PROGRAM Circuito_L4
VAR_INPUT
	Modo_Calibrar_L4: BOOL;
END_VAR
	
VAR
		fbBomba_L4 :Equipo_Motor_ATV320;
		ControlValv_ioLink_V1:ControlValv_ioLink;
		ControlValv_ioLink_V2: ControlValv_ioLink;
		ControlValv_ioLink_V3: ControlValv_ioLink;
		ControlValv_ioLink_V4: ControlValv_ioLink;
		Falla_L4_V1:BOOL;
		Falla_L4_V2:BOOL;
		Falla_L4_V3:BOOL;
		Falla_L4_V4:BOOL;
	Balanza_PU1_WT4: Balanza;
		dHS:DINT;
		TOF_calibradoIBC: TOF;
		TDemoraInyectar: TON;
		SetDemoraInyeccion: REAL;
	

	Volumen_L4: REAL;
	AuxVol: REAL;
	Total: REAL;
	auxIniCal: BOOL;
	Calculo_caudal_L4: Calculo_caudal;
	PID_L4_SP: REAL;
	PID_L4_PV: REAL;
	CorrecionCaudalxOffset_L4: CorrecionCaudalxOffset;
	tInyeccion: TON;
	PID_L4_manual: REAL;
	PID_L4: FB_PID;
	PID_L4_Kp: REAL := 0.1;
	PID_L4_Ti: REAL := 100;
	PID_L4_auto: BOOL;
	PID_L4_reset: BOOL;
	PID_L4_bMuerta: REAL := 5;
	Tiempo_seg_to_TIME_DemoraInyec: Tiempo_seg_to_TIME;
	AuxTDemoraInyec: TIME;
	Tiempo_TIME_to_seg_InyCal: Tiempo_TIME_to_seg;
	AuxInyCal:TIME;
	IniTotalFT2:REAL;
	Auxconsumo:REAL;
	ProductoAsociado: STRING;
	Lavagem_Circuito04: Lavagem;
	
END_VAR
VAR PERSISTENT
	UltimaCalibracao	:UDINT;	//Data e hora da ultima calibração
END_VAR
VAR // added by the converter: edge detectors and wires of the graphical bodies
    _w1, _w2, _w3, _w4, _w5, _w6, _w7, _w8, _w9, _w10, _w11, _w12, _w13 : BOOL;
    _ft1 : F_TRIG;
    _rt1, _rt2 : R_TRIG;
END_VAR

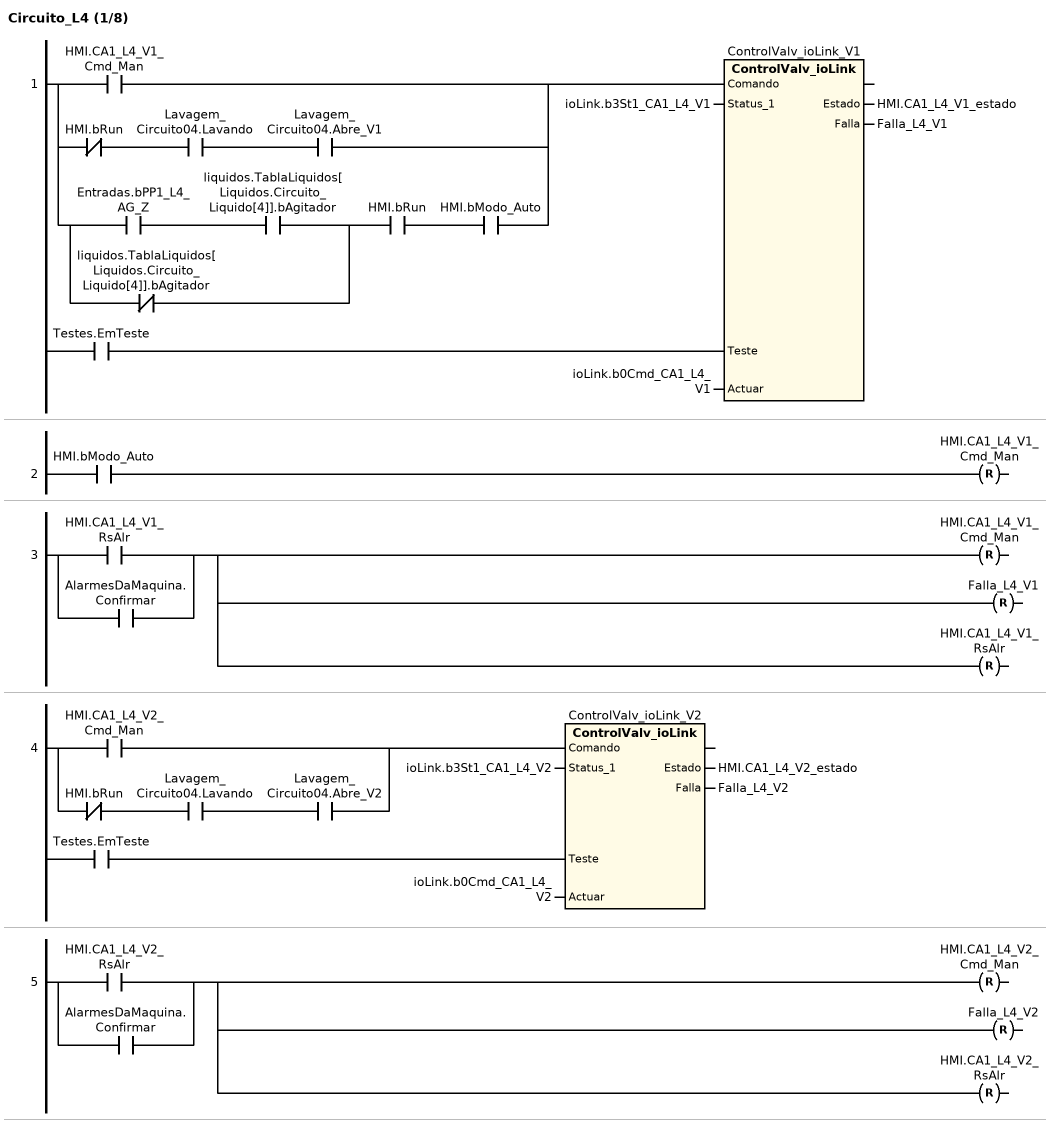
// NETWORK 1
ControlValv_ioLink_V1(
    Comando := HMI.CA1_L4_V1_Cmd_Man OR NOT HMI.bRun AND Lavagem_Circuito04.Lavando AND Lavagem_Circuito04.Abre_V1 OR (Entradas.bPP1_L4_AG_Z AND (liquidos.TablaLiquidos[Liquidos.Circuito_Liquido[4]].bAgitador) OR NOT (liquidos.TablaLiquidos[Liquidos.Circuito_Liquido[4]].bAgitador)) AND HMI.bRun AND HMI.bModo_Auto,
    Status_1 := ioLink.b3St1_CA1_L4_V1,
    Teste := Testes.EmTeste,
    Actuar := ioLink.b0Cmd_CA1_L4_V1,
    Estado => HMI.CA1_L4_V1_estado,
    Falla => Falla_L4_V1); // ControlValv_ioLink

// NETWORK 2
HMI.CA1_L4_V1_Cmd_Man R= HMI.bModo_Auto;

// NETWORK 3
_w1 := HMI.CA1_L4_V1_RsAlr OR AlarmesDaMaquina.Confirmar;
HMI.CA1_L4_V1_Cmd_Man R= _w1;
Falla_L4_V1 R= _w1;
HMI.CA1_L4_V1_RsAlr R= _w1;

// NETWORK 4
ControlValv_ioLink_V2(
    Comando := HMI.CA1_L4_V2_Cmd_Man OR NOT HMI.bRun AND Lavagem_Circuito04.Lavando AND Lavagem_Circuito04.Abre_V2,
    Status_1 := ioLink.b3St1_CA1_L4_V2,
    Teste := Testes.EmTeste,
    Actuar := ioLink.b0Cmd_CA1_L4_V2,
    Estado => HMI.CA1_L4_V2_estado,
    Falla => Falla_L4_V2); // ControlValv_ioLink

// NETWORK 5
_w2 := HMI.CA1_L4_V2_RsAlr OR AlarmesDaMaquina.Confirmar;
HMI.CA1_L4_V2_Cmd_Man R= _w2;
Falla_L4_V2 R= _w2;
HMI.CA1_L4_V2_RsAlr R= _w2;

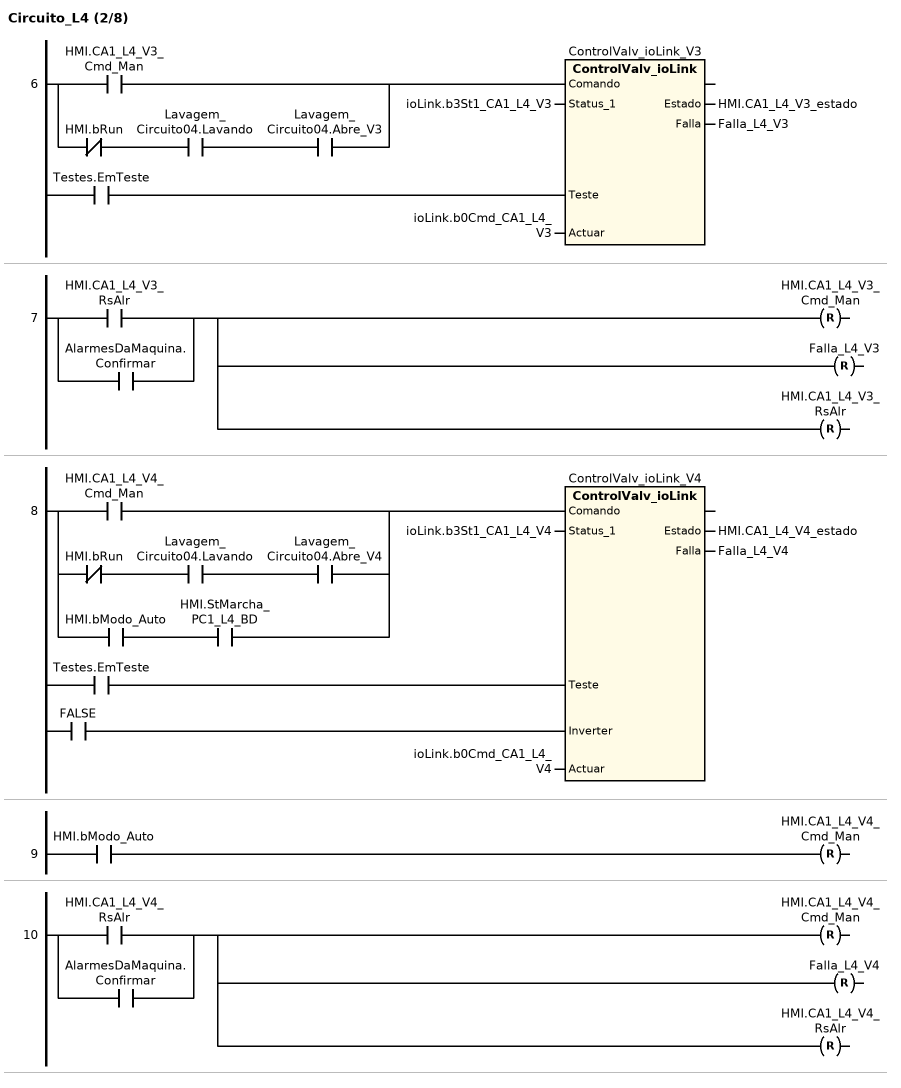
// NETWORK 6
ControlValv_ioLink_V3(
    Comando := HMI.CA1_L4_V3_Cmd_Man OR NOT HMI.bRun AND Lavagem_Circuito04.Lavando AND Lavagem_Circuito04.Abre_V3,
    Status_1 := ioLink.b3St1_CA1_L4_V3,
    Teste := Testes.EmTeste,
    Actuar := ioLink.b0Cmd_CA1_L4_V3,
    Estado => HMI.CA1_L4_V3_estado,
    Falla => Falla_L4_V3); // ControlValv_ioLink

// NETWORK 7
_w3 := HMI.CA1_L4_V3_RsAlr OR AlarmesDaMaquina.Confirmar;
HMI.CA1_L4_V3_Cmd_Man R= _w3;
Falla_L4_V3 R= _w3;
HMI.CA1_L4_V3_RsAlr R= _w3;

// NETWORK 8
ControlValv_ioLink_V4(
    Comando := HMI.CA1_L4_V4_Cmd_Man OR NOT HMI.bRun AND Lavagem_Circuito04.Lavando AND Lavagem_Circuito04.Abre_V4 OR HMI.bModo_Auto AND HMI.StMarcha_PC1_L4_BD,
    Status_1 := ioLink.b3St1_CA1_L4_V4,
    Teste := Testes.EmTeste,
    Inverter := FALSE,
    Actuar := ioLink.b0Cmd_CA1_L4_V4,
    Estado => HMI.CA1_L4_V4_estado,
    Falla => Falla_L4_V4); // ControlValv_ioLink

// NETWORK 9
HMI.CA1_L4_V4_Cmd_Man R= HMI.bModo_Auto;

// NETWORK 10
_w4 := HMI.CA1_L4_V4_RsAlr OR AlarmesDaMaquina.Confirmar;
HMI.CA1_L4_V4_Cmd_Man R= _w4;
Falla_L4_V4 R= _w4;
HMI.CA1_L4_V4_RsAlr R= _w4;

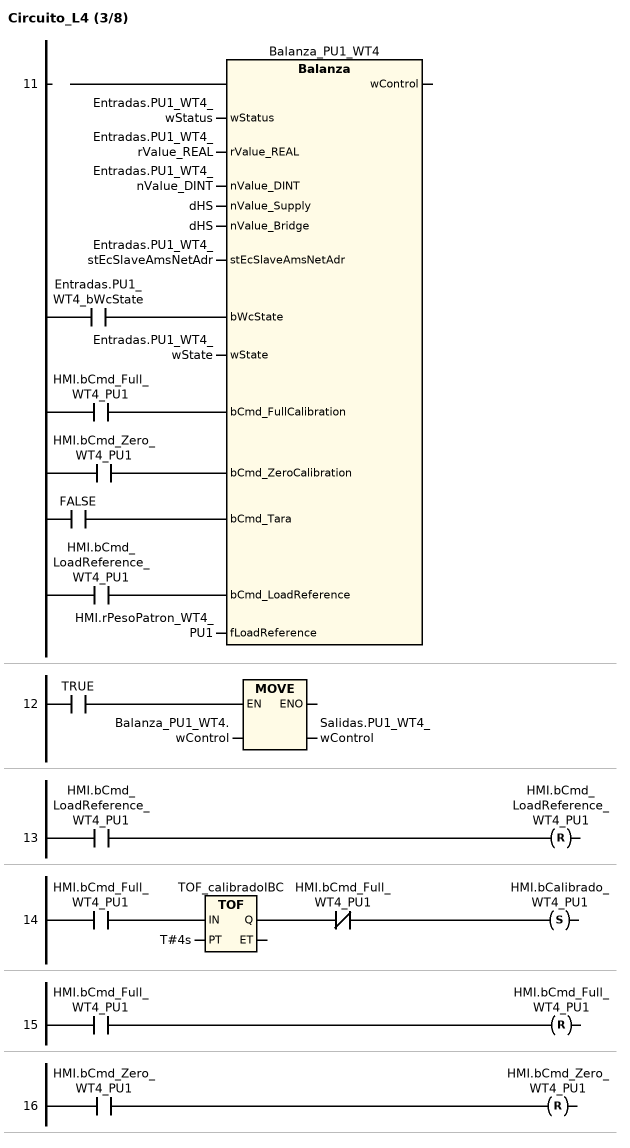
// NETWORK 11
Balanza_PU1_WT4(
    wStatus := Entradas.PU1_WT4_wStatus,
    rValue_REAL := Entradas.PU1_WT4_rValue_REAL,
    nValue_DINT := Entradas.PU1_WT4_nValue_DINT,
    nValue_Supply := dHS,
    nValue_Bridge := dHS,
    stEcSlaveAmsNetAdr := Entradas.PU1_WT4_stEcSlaveAmsNetAdr,
    bWcState := Entradas.PU1_WT4_bWcState,
    wState := Entradas.PU1_WT4_wState,
    bCmd_FullCalibration := HMI.bCmd_Full_WT4_PU1,
    bCmd_ZeroCalibration := HMI.bCmd_Zero_WT4_PU1,
    bCmd_Tara := FALSE,
    bCmd_LoadReference := HMI.bCmd_LoadReference_WT4_PU1,
    fLoadReference := HMI.rPesoPatron_WT4_PU1); // Balanza

// NETWORK 12
Salidas.PU1_WT4_wControl := Balanza_PU1_WT4.wControl;

// NETWORK 13
HMI.bCmd_LoadReference_WT4_PU1 R= HMI.bCmd_LoadReference_WT4_PU1;

// NETWORK 14
TOF_calibradoIBC(IN := HMI.bCmd_Full_WT4_PU1, PT := T#4s); // TOF
HMI.bCalibrado_WT4_PU1 S= TOF_calibradoIBC.Q AND NOT HMI.bCmd_Full_WT4_PU1;

// NETWORK 15
HMI.bCmd_Full_WT4_PU1 R= HMI.bCmd_Full_WT4_PU1;

// NETWORK 16
HMI.bCmd_Zero_WT4_PU1 R= HMI.bCmd_Zero_WT4_PU1;

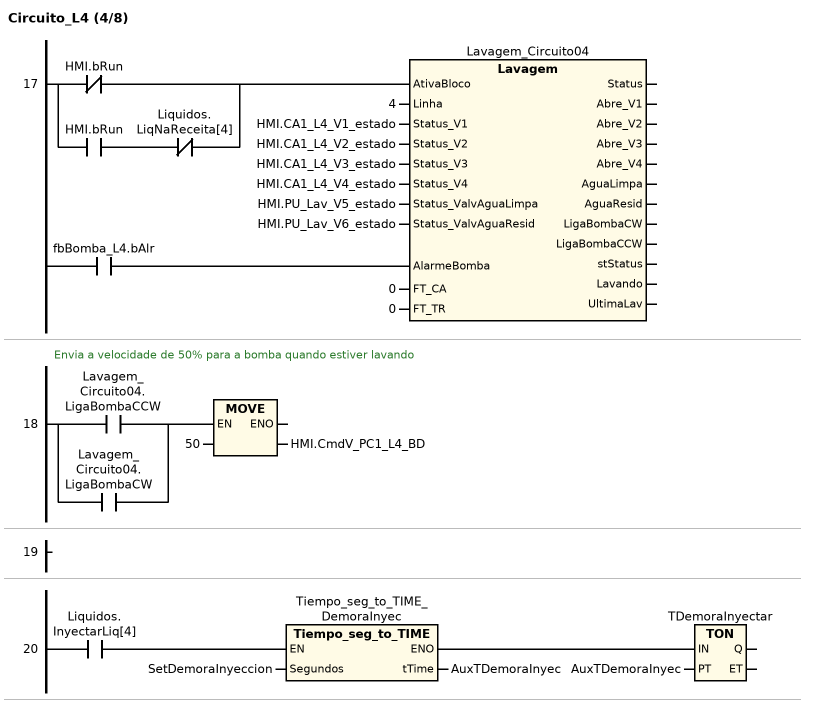
// NETWORK 17
Lavagem_Circuito04(
    AtivaBloco := NOT HMI.bRun OR HMI.bRun AND NOT Liquidos.LiqNaReceita[4],
    Linha := 4,
    Status_V1 := HMI.CA1_L4_V1_estado,
    Status_V2 := HMI.CA1_L4_V2_estado,
    Status_V3 := HMI.CA1_L4_V3_estado,
    Status_V4 := HMI.CA1_L4_V4_estado,
    Status_ValvAguaLimpa := HMI.PU_Lav_V5_estado,
    Status_ValvAguaResid := HMI.PU_Lav_V6_estado,
    AlarmeBomba := fbBomba_L4.bAlr,
    FT_CA := 0,
    FT_TR := 0); // Lavagem

// NETWORK 18
// Envia a velocidade de 50% para a bomba quando estiver lavando
IF Lavagem_Circuito04.LigaBombaCCW OR Lavagem_Circuito04.LigaBombaCW THEN HMI.CmdV_PC1_L4_BD := 50; END_IF

// NETWORK 19

// NETWORK 20
_w5 := Liquidos.InyectarLiq[4];
IF _w5 THEN
    Tiempo_seg_to_TIME_DemoraInyec(Segundos := SetDemoraInyeccion, tTime => AuxTDemoraInyec); // Tiempo_seg_to_TIME
END_IF
TDemoraInyectar(IN := _w5, PT := AuxTDemoraInyec); // TON

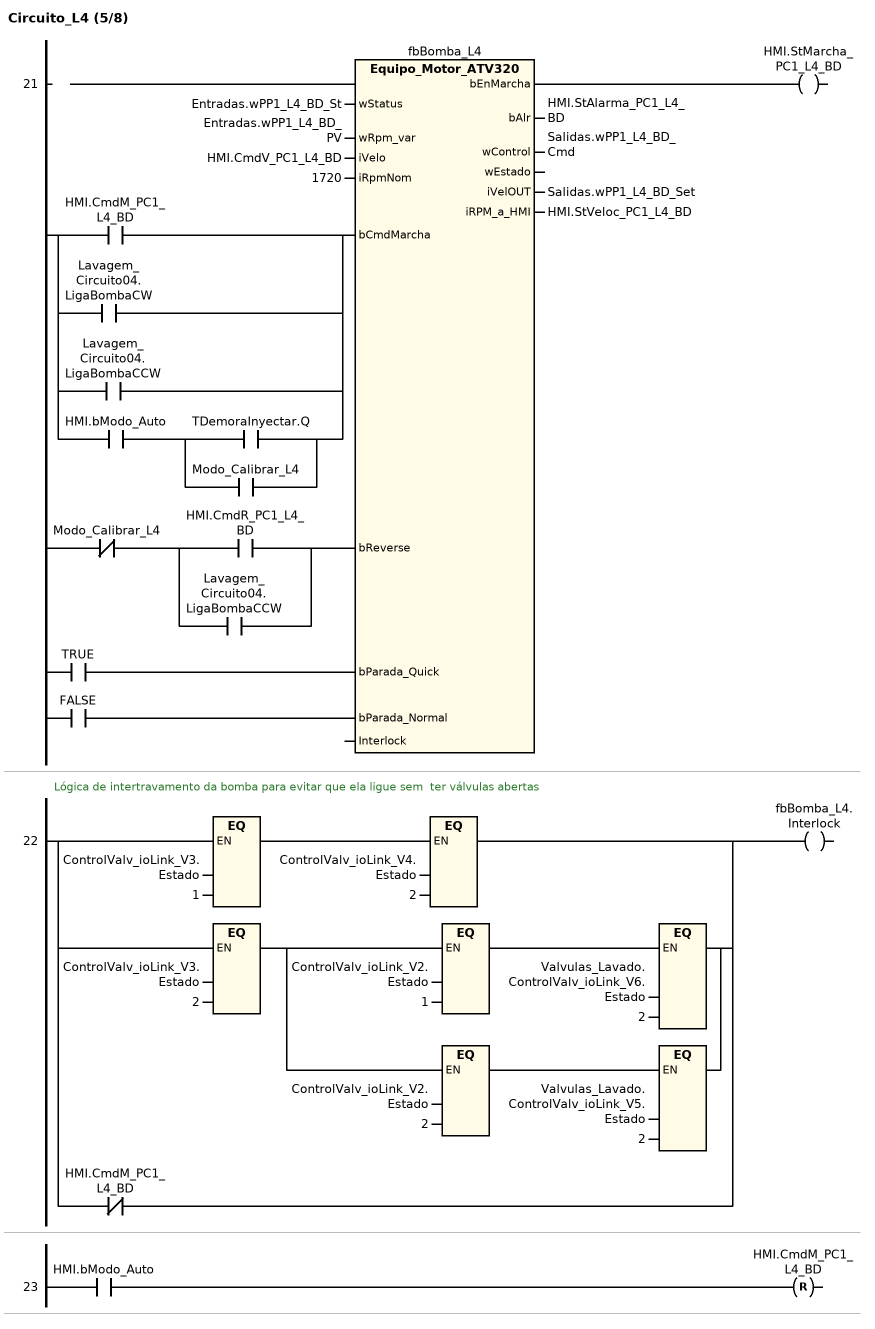
// NETWORK 21
fbBomba_L4(
    wStatus := Entradas.wPP1_L4_BD_St,
    wRpm_var := Entradas.wPP1_L4_BD_PV,
    iVelo := HMI.CmdV_PC1_L4_BD,
    iRpmNom := 1720,
    bCmdMarcha := HMI.CmdM_PC1_L4_BD OR Lavagem_Circuito04.LigaBombaCW OR Lavagem_Circuito04.LigaBombaCCW OR HMI.bModo_Auto AND (TDemoraInyectar.Q OR Modo_Calibrar_L4),
    bReverse := NOT Modo_Calibrar_L4 AND (HMI.CmdR_PC1_L4_BD OR Lavagem_Circuito04.LigaBombaCCW),
    bParada_Quick := TRUE,
    bParada_Normal := FALSE,
    bAlr => HMI.StAlarma_PC1_L4_BD,
    wControl => Salidas.wPP1_L4_BD_Cmd,
    iVelOUT => Salidas.wPP1_L4_BD_Set,
    iRPM_a_HMI => HMI.StVeloc_PC1_L4_BD); // Equipo_Motor_ATV320
HMI.StMarcha_PC1_L4_BD := fbBomba_L4.bEnMarcha;

// NETWORK 22
// Lógica de intertravamento da bomba para evitar que ela ligue sem  ter válvulas abertas
_w6 := NOT HMI.CmdM_PC1_L4_BD;
IF NOT _w6 THEN
    _w7 := ControlValv_ioLink_V3.Estado = 2;
    _w6 := ControlValv_ioLink_V3.Estado = 1 AND ControlValv_ioLink_V4.Estado = 2 OR (_w7 AND ControlValv_ioLink_V2.Estado = 1 AND Valvulas_Lavado.ControlValv_ioLink_V6.Estado = 2 OR _w7 AND ControlValv_ioLink_V2.Estado = 2 AND Valvulas_Lavado.ControlValv_ioLink_V5.Estado = 2);
END_IF
fbBomba_L4.Interlock := _w6;

// NETWORK 23
HMI.CmdM_PC1_L4_BD R= HMI.bModo_Auto;

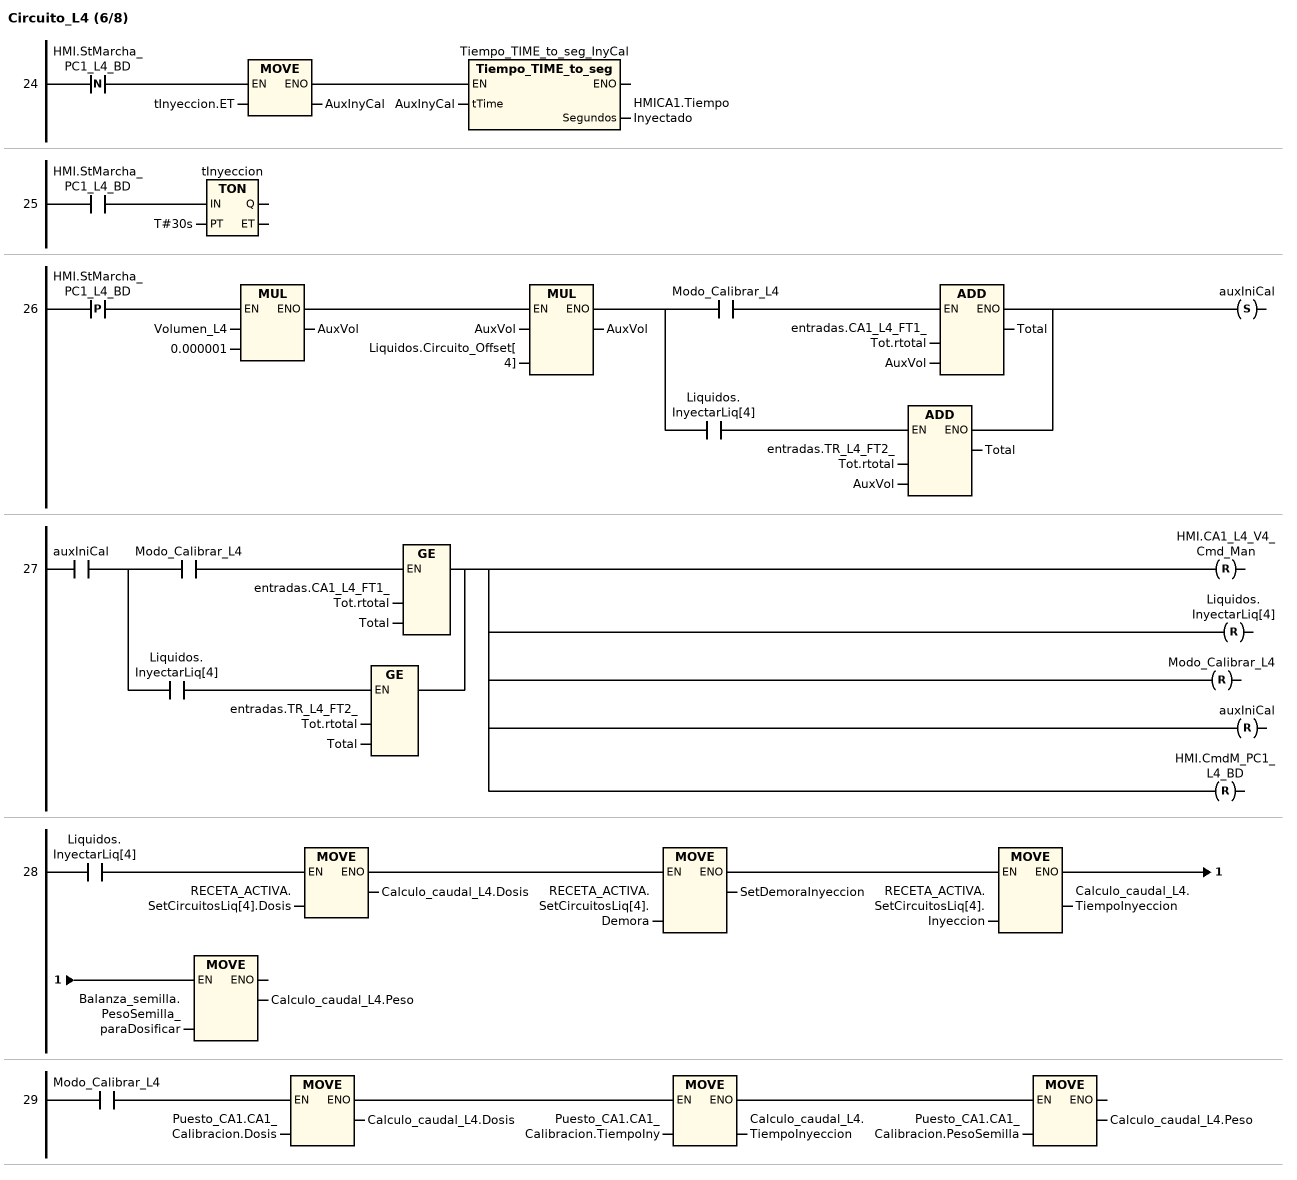
// NETWORK 24
_ft1(CLK := HMI.StMarcha_PC1_L4_BD);
_w8 := _ft1.Q;
IF _w8 THEN AuxInyCal := tInyeccion.ET; END_IF
IF _w8 THEN
    Tiempo_TIME_to_seg_InyCal(tTime := AuxInyCal, Segundos => HMICA1.TiempoInyectado); // Tiempo_TIME_to_seg
END_IF

// NETWORK 25
tInyeccion(IN := HMI.StMarcha_PC1_L4_BD, PT := T#30s); // TON

// NETWORK 26
_rt1(CLK := HMI.StMarcha_PC1_L4_BD);
_w9 := _rt1.Q;
IF _w9 THEN AuxVol := Volumen_L4 * 0.000001; END_IF
IF _w9 THEN AuxVol := AuxVol * Liquidos.Circuito_Offset[4]; END_IF
IF _w9 AND Modo_Calibrar_L4 THEN Total := entradas.CA1_L4_FT1_Tot.rtotal + AuxVol; END_IF
IF _w9 AND Liquidos.InyectarLiq[4] THEN Total := entradas.TR_L4_FT2_Tot.rtotal + AuxVol; END_IF
auxIniCal S= _w9 AND Modo_Calibrar_L4 OR _w9 AND Liquidos.InyectarLiq[4];

// NETWORK 27
_w10 := auxIniCal AND Modo_Calibrar_L4 AND entradas.CA1_L4_FT1_Tot.rtotal >= Total OR auxIniCal AND Liquidos.InyectarLiq[4] AND entradas.TR_L4_FT2_Tot.rtotal >= Total;
HMI.CA1_L4_V4_Cmd_Man R= _w10;
Liquidos.InyectarLiq[4] R= _w10;
Modo_Calibrar_L4 R= _w10;
auxIniCal R= _w10;
HMI.CmdM_PC1_L4_BD R= _w10;

// NETWORK 28
_w11 := Liquidos.InyectarLiq[4];
IF _w11 THEN Calculo_caudal_L4.Dosis := RECETA_ACTIVA.SetCircuitosLiq[4].Dosis; END_IF
IF _w11 THEN SetDemoraInyeccion := RECETA_ACTIVA.SetCircuitosLiq[4].Demora; END_IF
IF _w11 THEN Calculo_caudal_L4.TiempoInyeccion := RECETA_ACTIVA.SetCircuitosLiq[4].Inyeccion; END_IF
IF _w11 THEN Calculo_caudal_L4.Peso := Balanza_semilla.PesoSemilla_paraDosificar; END_IF

// NETWORK 29
_w12 := Modo_Calibrar_L4;
IF _w12 THEN Calculo_caudal_L4.Dosis := Puesto_CA1.CA1_Calibracion.Dosis; END_IF
IF _w12 THEN Calculo_caudal_L4.TiempoInyeccion := Puesto_CA1.CA1_Calibracion.TiempoIny; END_IF
IF _w12 THEN Calculo_caudal_L4.Peso := Puesto_CA1.CA1_Calibracion.PesoSemilla; END_IF

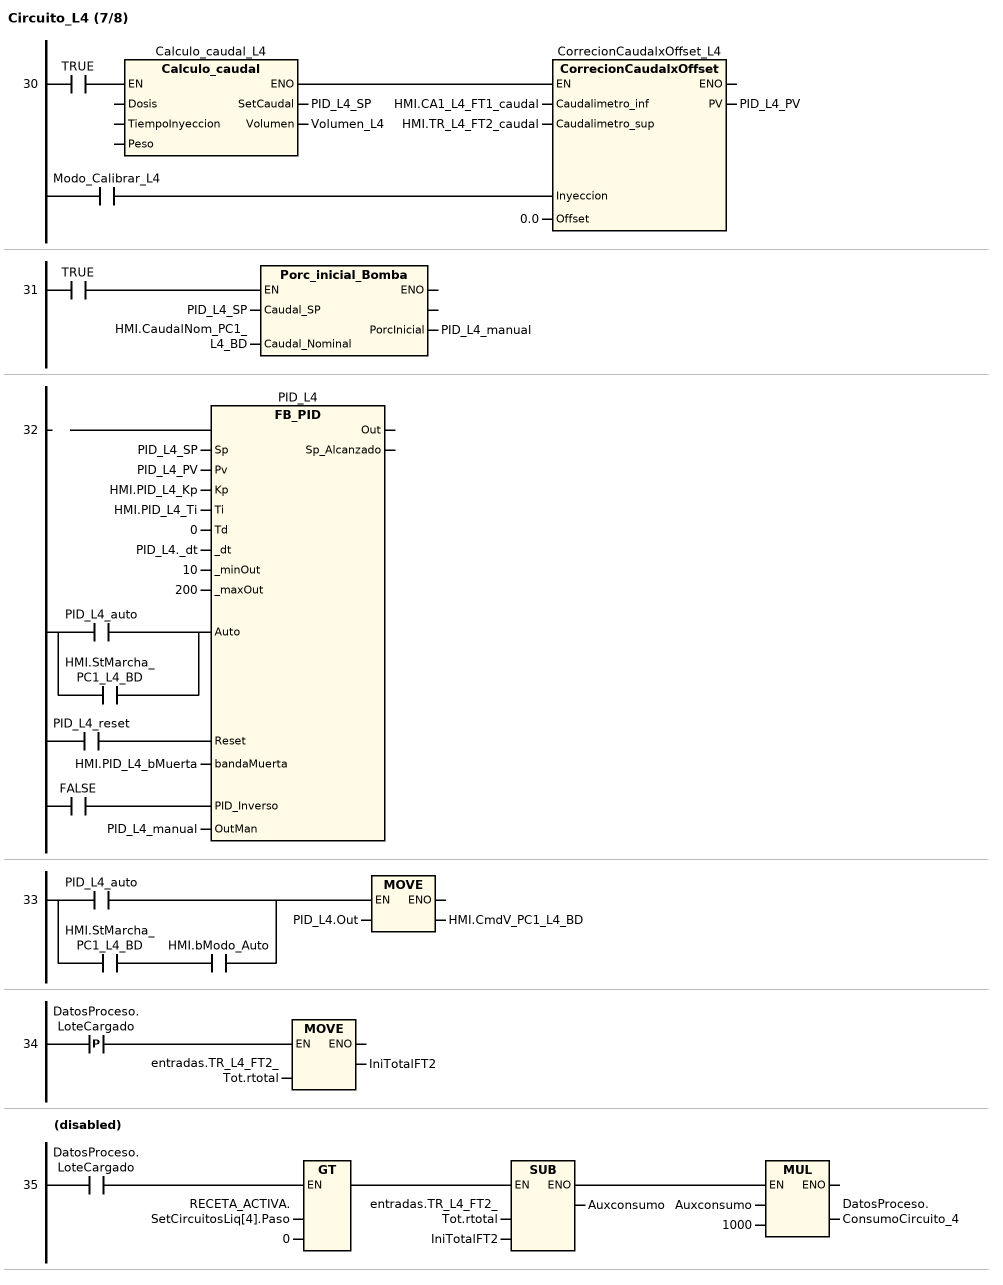
// NETWORK 30
Calculo_caudal_L4(SetCaudal => PID_L4_SP, Volumen => Volumen_L4); // Calculo_caudal
CorrecionCaudalxOffset_L4(
    Caudalimetro_inf := HMI.CA1_L4_FT1_caudal,
    Caudalimetro_sup := HMI.TR_L4_FT2_caudal,
    Inyeccion := Modo_Calibrar_L4,
    Offset := 0.0,
    PV => PID_L4_PV); // CorrecionCaudalxOffset

// NETWORK 31
Porc_inicial_Bomba(Caudal_SP := PID_L4_SP, Caudal_Nominal := HMI.CaudalNom_PC1_L4_BD, PorcInicial => PID_L4_manual);

// NETWORK 32
PID_L4(
    Sp := PID_L4_SP,
    Pv := PID_L4_PV,
    Kp := HMI.PID_L4_Kp,
    Ti := HMI.PID_L4_Ti,
    Td := 0,
    _dt := PID_L4._dt,
    _minOut := 10,
    _maxOut := 200,
    Auto := PID_L4_auto OR HMI.StMarcha_PC1_L4_BD,
    Reset := PID_L4_reset,
    bandaMuerta := HMI.PID_L4_bMuerta,
    PID_Inverso := FALSE,
    OutMan := PID_L4_manual); // FB_PID

// NETWORK 33
IF PID_L4_auto OR HMI.StMarcha_PC1_L4_BD AND HMI.bModo_Auto THEN HMI.CmdV_PC1_L4_BD := PID_L4.Out; END_IF

// NETWORK 34
_rt2(CLK := DatosProceso.LoteCargado);
IF _rt2.Q THEN IniTotalFT2 := entradas.TR_L4_FT2_Tot.rtotal; END_IF

// NETWORK 35 (disabled)
// _w13 := DatosProceso.LoteCargado AND RECETA_ACTIVA.SetCircuitosLiq[4].Paso > 0;
// IF _w13 THEN Auxconsumo := entradas.TR_L4_FT2_Tot.rtotal - IniTotalFT2; END_IF
// IF _w13 THEN DatosProceso.ConsumoCircuito_4 := Auxconsumo * 1000; END_IF

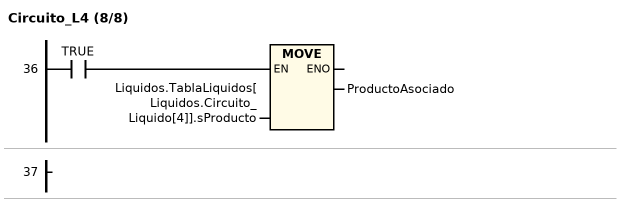
// NETWORK 36
ProductoAsociado := Liquidos.TablaLiquidos[Liquidos.Circuito_Liquido[4]].sProducto;

// NETWORK 37

END_PROGRAM

(* stored: Version 1.1.0.1, ProductVersion 3.1.4024.14
   POU Circuito_L4: Id {9d4cdb36-8d27-4600-8e01-71ec27e8d612}, SpecialFunc None *)
